Staubli VAL3: onStart.pgx

public program onStart(string& x_sItem[])
begin
  //
  // ANALOGIC VALUE
  //
  // default use the COUNTER
  call saveInOut:setOutput(10)
  call saveInOut:setInput(10)
  // MODBUS
  call saveInOut:setOutput(11)
  call saveInOut:setInput(11)
  // USER
  call saveInOut:setOutput(12)
  call saveInOut:setInput(12)
  // REMIO
  call saveInOut:setOutput(13)
  call saveInOut:setInput(13)
  // Other
  call saveInOut:setOutput(14)
  call saveInOut:setInput(14)
end
